FUNCTION_BLOCK FB_CSVEventStorage IMPLEMENTS I_CSVEventStorage
VAR
	fbFileOpen : FB_FileOpen := (sPathName := 'C:\Event.log', nMode := FOPEN_MODEAPPEND OR FOPEN_MODETEXT);
	fbFileClose: FB_FileClose;
	fbFilePuts : FB_FilePuts;
	eState : (FILE_OPEN_TRIGGER, FILE_OPEN, WAIT_FOR_EVENT, WRITE_EVENT_TRIGGER, WRITE_EVENT,FILE_CLOSE_TRIGGER, FILE_CLOSE, ERROR);
	stEventToBeWrittenToFile : ST_Event;
	CSVStr : T_MaxString;	
END_VAR

 CASE eState OF
	 FILE_OPEN_TRIGGER:
	 	fbFileOpen(bExecute := TRUE);
		eState := FILE_OPEN;
		
	 FILE_OPEN:
	 	fbFileOpen(bExecute := FALSE);
	 	IF fbFileOpen.bError THEN
			eState := ERROR;
		ELSIF NOT fbFileOpen.bBusy AND fbFileOpen.hFile <> 0 THEN
			eState := WAIT_FOR_EVENT;
		END_IF		
		
	WAIT_FOR_EVENT:
		//Do Nothing
		
	WRITE_EVENT_TRIGGER:
	CSVStr := CSVCompatibleString(stEventToBeWrittenToFile);
	fbFilePuts(bExecute:=TRUE, sLine :=CSVStr, hFile := fbFileOpen.hFile);
	eState := WRITE_EVENT;	
	
	WRITE_EVENT:
	fbFilePuts(bExecute:=FALSE);
	IF fbFilePuts.bError THEN
		eState := ERROR;
	ELSIF NOT fbFilePuts.bBusy THEN
		eState := FILE_CLOSE_TRIGGER;
	END_IF	
	
	FILE_CLOSE_TRIGGER:
		fbFileClose(bExecute:= TRUE, hFile:= fbFileOpen.hFile);
		eState := FILE_CLOSE; 
	
	FILE_CLOSE:
		fbFileClose(bExecute:= FALSE);
		IF fbFileClose.bError THEN
			eState:= ERROR;
		ELSIF NOT fbFileClose.bBusy THEN
			eState := FILE_OPEN_TRIGGER;
		END_IF
		
	ERROR:
		//To do	 	
 END_CASE

METHOD PRIVATE CSVCompatibleString : T_MaxString
VAR_INPUT
	stEvent : REFERENCE TO ST_Event;
END_VAR
VAR
	TempStr : T_MaxString;
END_VAR
TempStr := TO_STRING(stEvent.eEventType);
TempStr := CONCAT(STR1 := TempStr, STR2 := ',');
TempStr := CONCAT(STR1 := TempStr, STR2 := TO_STRING(stEvent.eEventSeverity));
TempStr := CONCAT(STR1 := TempStr, STR2 := ',');
TempStr := CONCAT(STR1 := TempStr, STR2 := TO_STRING(stEvent.nEventDefinition));
TempStr := CONCAT(STR1 := TempStr, STR2 := ',');
TempStr := CONCAT(STR1 := TempStr, STR2 := stEvent.sEventMessage);
TempStr := CONCAT(STR1 := TempStr, STR2 := ',');
TempStr := CONCAT(STR1 := TempStr, STR2 := TO_STRING(stEvent.tTimeStamp));
TempStr := CONCAT(STR1 := TempStr, STR2 := '$n');

CSVCompatibleString := TempStr;
END_METHOD

METHOD StoreEvent
VAR_INPUT
	stEvent	: ST_Event;
END_VAR
IF eState = WAIT_FOR_EVENT THEN
	eState := WRITE_EVENT_TRIGGER;
	stEventToBeWrittenToFile := stEvent;
END_IF
END_METHOD

END_FUNCTION_BLOCK

(* stored: Version 1.1.0.1, ProductVersion 3.1.4024.9
   POU FB_CSVEventStorage: Id {4607d0b1-970b-4d0f-bcad-4a4b0c2eaa5d}, SpecialFunc None
   Method CSVCompatibleString: Id {e965b2be-c955-4662-bfc3-ff9841c3ab81}
   Method StoreEvent: Id {1c687bfc-bfa1-465f-b608-95184f3e00b0} *)
